TEXTLIST TL_E_CTRL_MOVER
  0 = 'MOVER_NULL'
  1 = 'MOVER_ENABLE'
  2 = 'MOVER_DISABLE'
  4 = 'MOVER_MOVE_TO_POS_CA'
  5 = 'MOVER_SEND_TO_POS_CA'
  6 = 'MOVER_HALT'
  7 = 'MOVER_GEAR_IN'
  8 = 'MOVER_GEAR_IN_POS_CA'
  9 = 'MOVER_GEAR_OUT'
  10 = 'MOVER_RESET'
  3 = 'MOVER_MOVE_TO_POS'
   = ''
END_TEXTLIST

(* stored: Version 1.1.0.1
   TextList TL_E_CTRL_MOVER: Id {382d03bc-16b1-4fa2-aebc-40883fed74e1} *)
